// TIA Portal V20 export
DATA_BLOCK "I_Data"   // DB15
{ S7_Optimized_Access := 'FALSE' }
   VAR
      Data_IN : Struct
         Data_I_1 : Int := 1;
         Data_I_2 : Int := 2;
         Data_I_3 : Int := 3;
         Data_I_4 : Int := 4;
         Data_I_5 : Int := 5;
         Data_I_6 : Int := 6;
         Data_I_7 : Int := 7;
         Data_I_8 : Int := 8;
      END_STRUCT;
   END_VAR
BEGIN
END_DATA_BLOCK
